FUNCTION_BLOCK FB_ElementLUT EXTENDS FB_Fallible IMPLEMENTS I_StringLookupElement
VAR
    iAtomicMassLUT : I_StringLookupLREAL;
    iAtomicNumberLUT : I_StringLookupINT;
    iDensityLUT : I_StringLookupLREAL;
END_VAR


METHOD FB_Init: BOOL
VAR_INPUT
    bInitRetains: BOOL; // TRUE: the retain variables are initialized (reset warm / reset cold)
    bInCopyCode: BOOL;  // TRUE: the instance will be copied to the copy code afterward (online change)

    iAtomicMassLUT : I_StringLookupLREAL;
    iAtomicNumberLUT : I_StringLookupINT;
    iDensityLUT : I_StringLookupLREAL;
END_VAR

THIS^.iAtomicMassLUT := iAtomicMassLUT;
THIS^.iAtomicNumberLUT := iAtomicNumberLUT;
THIS^.iDensityLUT := iDensityLUT;
END_METHOD


METHOD LookupAtomicMass : LREAL
VAR_INPUT
    sLookup	: STRING;
END_VAR
VAR
    fAtomicMass : LREAL;
END_VAR

fAtomicMass := iAtomicMassLUT.Lookup(sLookup := sLookup);

IF iAtomicMassLUT.GetError() THEN
    SetError(
        sMsg := CONCAT('The atomic mass lookup table has an error: ',
        iAtomicMassLUT.GetErrorMsg())
    );
    RETURN;
END_IF

LookupAtomicMass := fAtomicMass;
END_METHOD


METHOD LookupAtomicNumber : INT
VAR_INPUT
    sLookup	: STRING;
END_VAR
VAR
    nAtomicNumber : INT;
END_VAR

LookupAtomicNumber := -1;

nAtomicNumber := iAtomicNumberLUT.Lookup(sLookup := sLookup);

IF iAtomicNumberLUT.GetError() THEN
    SetError(
        sMsg := CONCAT('The atomic number lookup table has an error: ',
        iAtomicNumberLUT.GetErrorMsg())
    );
    RETURN;
END_IF

LookupAtomicNumber := nAtomicNumber;
END_METHOD

{warning 'Add method implementation '}
METHOD LookupDensity : LREAL
VAR_INPUT
    sLookup	: STRING;
END_VAR
VAR
    fDensity : LREAL;
END_VAR

fDensity := iDensityLUT.Lookup(sLookup := sLookup);

IF iDensityLUT.GetError() THEN
    SetError(
        sMsg := CONCAT('The density lookup table has an error: ',
        iDensityLUT.GetErrorMsg())
    );
    RETURN;
END_IF

LookupDensity := fDensity;
END_METHOD

END_FUNCTION_BLOCK

(* stored: Version 1.1.0.1
   POU FB_ElementLUT: Id {396e148e-5a54-4e0f-be5e-d5ad59e7e763}, SpecialFunc None
   Method FB_Init: Id {e170e441-4319-4285-be2c-da9c65660aea}
   Method LookupAtomicMass: Id {b49da3c3-29e7-4735-b051-4bef81174655}
   Method LookupAtomicNumber: Id {9aa2ed00-c722-4992-b0e5-7489d0c70f8e}
   Method LookupDensity: Id {b0ef6550-2f85-4569-94b6-5ef5f47fa201} *)
